// TwinCAT 3 PLC project safety
// ProgramVersion: 3.1.4024.0
// libraries:
//   Tc2_Standard, * (Beckhoff Automation GmbH)
//   Tc2_System, * (Beckhoff Automation GmbH)
//   Tc3_Module, * (Beckhoff Automation GmbH)
// project tree:
//   / PlcTask.TcTTO
//   POUs/ MAIN.TcPOU
// real-time tasks:
//   TASK Safety: cycle T#5ms, priority 6, ADS port 350
//   TASK StateMachine: cycle T#1ms, priority 4, ADS port 351
// I/O:
//   DEVICE Device 5 (EtherCAT), AmsNetId 192.168.0.231.6.1
//     Term 1 (EK1100) [EK1100 EtherCAT Coupler (2A E-Bus)]
//       Term 2 (EL3702) [EL3702 2Ch. Ana. Input +/-10V, DIFF, Oversample]
//       Term 3 (EL3702) [EL3702 2Ch. Ana. Input +/-10V, DIFF, Oversample]
//       Term 4 (EL3702) [EL3702 2Ch. Ana. Input +/-10V, DIFF, Oversample]
//       Term 5 (EL1004) [EL1004 4Ch. Dig. Input 24V, 3ms]
//       Term 6 (EL1004) [EL1004 4Ch. Dig. Input 24V, 3ms]
//       Term 7 (EL2004) [EL2004 4Ch. Dig. Output 24V, 0.5A]
//       Term 8 (EL2004) [EL2004 4Ch. Dig. Output 24V, 0.5A]
//       Term 9 (EL6910) [EL6910, TwinSAFE PLC]
//       Term 10 (EL1904) [EL1904, 4 Ch. Safety Input 24V, TwinSAFE]
//         modules: Module 1 (FSOES)
//       Term 12 (EL9011) [EL9011 End Terminal]
// variable links:
//   Device 5 (EtherCAT) <-> Device 5 (EtherCAT)/Term 1 (EK1100)/Term 10 (EL1904)
//     Term 1 (EK1100)/Term 9 (EL6910)/ConnectionOutputs/Message_3 RxPDO <-> Module 1 (FSOES)/TxPDO/FSOE
//   Device 5 (EtherCAT) <-> Device 5 (EtherCAT)/Term 1 (EK1100)/Term 5 (EL1004)
//     Term 1 (EK1100)/Term 9 (EL6910)/StandardOutputs/Standard In Var 1 <-> Channel 2/Input
//   Device 5 (EtherCAT) <-> Device 5 (EtherCAT)/Term 1 (EK1100)/Term 9 (EL6910)
//     Term 1 (EK1100)/Term 10 (EL1904)/Module 1 (FSOES)/RxPDO/FSOE <-> ConnectionInputs/Message_3 TxPDO
//   safety/safety Instance <-> Device 5 (EtherCAT)/Term 1 (EK1100)/Term 8 (EL2004)
//     PlcTask Outputs/MAIN.b_LED <-> Channel 2/Output
//   safety/safety Instance <-> Device 5 (EtherCAT)/Term 1 (EK1100)/Term 9 (EL6910)
//     PlcTask Inputs/MAIN.b_ESTOPgen <-> StandardInputs/Standard Out Var 5
//     PlcTask Inputs/MAIN.b_SafetyState <-> StandardInputs/Standard Out Var 4
//     PlcTask Outputs/MAIN.b_Run <-> StandardOutputs/Standard In Var 2
//   safety/safety Instance <-> state_machine_prj/state_machine_prj Instance
//     PlcTask Outputs/MAIN.b_ESTOPout <-> PlcTask Inputs/MAIN.b_estop
//     PlcTask Outputs/MAIN.b_LED <-> PlcTask Inputs/MAIN.b_resetLed
//     PlcTask Outputs/MAIN.b_SafetyStateOut <-> PlcTask Inputs/MAIN.b_reset
//   state_machine_prj/state_machine_prj Instance <-> Device 5 (EtherCAT)/Term 1 (EK1100)/Term 2 (EL3702)
//     PlcTask Inputs/MAIN.n_A_sensors[0] <-> Ch2 Sample 0/Ch2 Value
//     PlcTask Inputs/MAIN.n_A_sensors[1] <-> Ch1 Sample 0/Ch1 Value
//   state_machine_prj/state_machine_prj Instance <-> Device 5 (EtherCAT)/Term 1 (EK1100)/Term 4 (EL3702)
//     PlcTask Inputs/MAIN.n_V_sensors[0] <-> Ch1 Sample 0/Ch1 Value
//     PlcTask Inputs/MAIN.n_V_sensors[1] <-> Ch2 Sample 0/Ch2 Value
//   state_machine_prj/state_machine_prj Instance <-> Device 5 (EtherCAT)/Term 1 (EK1100)/Term 6 (EL1004)
//     PlcTask Inputs/MAIN.b_bypass_contactors_fb[0] <-> Channel 3/Input
//     PlcTask Inputs/MAIN.b_bypass_contactors_fb[1] <-> Channel 4/Input
//     PlcTask Inputs/MAIN.b_main_contactors_fb[0] <-> Channel 1/Input
//     PlcTask Inputs/MAIN.b_main_contactors_fb[1] <-> Channel 2/Input
//   state_machine_prj/state_machine_prj Instance <-> Device 5 (EtherCAT)/Term 1 (EK1100)/Term 7 (EL2004)
//     PlcTask Outputs/MAIN.b_bypass_contactors[0] <-> Channel 3/Output
//     PlcTask Outputs/MAIN.b_bypass_contactors[1] <-> Channel 4/Output
//     PlcTask Outputs/MAIN.b_main_contactors[0] <-> Channel 1/Output
//     PlcTask Outputs/MAIN.b_main_contactors[1] <-> Channel 2/Output

CONFIGURATION safety
    RESOURCE PLC ON TwinCAT3
        TASK PlcTask(INTERVAL := T#5ms, PRIORITY := 6);
        PROGRAM MAIN WITH PlcTask : MAIN;
    END_RESOURCE
END_CONFIGURATION

// ---- POUs/MAIN.TcPOU
PROGRAM MAIN
VAR	
	b_Run 				AT %Q* 		: BOOL := TRUE;
	b_LED 		 		AT %Q* 		: BOOL;
	b_SafetyStateOut 	AT %Q*		: BOOL;
	b_ESTOPout			AT %Q*		: BOOL;
	
	b_SafetyState		AT %I*		: BOOL;
	b_ESTOPgen			AT %I*		: BOOL;  		
	
	t_blkLED 						: TON;
	
	n_idx 							: INT;
END_VAR

// Blinking LED
IF NOT(b_SafetyState) AND NOT(b_ESTOPgen) THEN
	b_LED := TRUE;
ELSIF NOT(b_SafetyState) AND b_ESTOPgen THEN
	t_blkLED(IN := NOT(t_blkLED.Q), PT := T#2S);
	b_LED := t_blkLED.ET > T#1S;
ELSE
	b_LED := FALSE;
	t_blkLED(IN := FALSE);
END_IF

b_SafetyStateOut := b_SafetyState;
b_ESTOPout := b_ESTOPgen;

END_PROGRAM
